{attribute 'enable_dynamic_creation'}
FUNCTION_BLOCK Serializable
VAR_INPUT
	pSubclassPointer : POINTER TO BYTE;
	nObjectSize : UDINT;
END_VAR
VAR_OUTPUT
	nWrittenBytes : UDINT;
END_VAR

METHOD Desirialize : POINTER TO BYTE;
VAR_INPUT
	 pSerialObject : POINTER TO BYTE;
END_VAR
MEMCPY(pSubclassPointer,pSerialObject,nObjectSize);
Desirialize := pSerialObject;
END_METHOD

METHOD Serialize : POINTER TO BYTE;
VAR_INPUT
END_VAR
Serialize := __NEW(BYTE,nObjectSize);
nWrittenBytes := MEMCPY(Serialize,pSubclassPointer ,nObjectSize);
END_METHOD

END_FUNCTION_BLOCK

(* stored: Version 1.1.0.1, ProductVersion 3.1.4024.2
   POU Serializable: Id {bf08be08-f416-4660-a172-8d54c48fb818}, SpecialFunc None
   Method Desirialize: Id {30347d4a-649e-49b4-b8f8-f206c96a3145}
   Method Serialize: Id {756b9a90-8f53-46bd-9d89-e8e40b346001} *)
